INTERFACE I_Disposer

METHOD Dispose
VAR_INPUT
	Source : I_WritableData;
END_VAR
END_METHOD

END_INTERFACE

(* stored: Version 1.1.0.1, ProductVersion 3.1.4024.12
   Itf I_Disposer: Id {4efb882e-a074-012a-0db9-6825328cb0ff}
   Method Dispose: Id {9aa1e6b5-0262-094e-3ecb-e00254fe3512} *)
